(* PLC project Unnamed, Unknown Unnamed 1 *)
(* stored: creationDateTime 2023-03-10T10:37:17, modificationDateTime 2023-03-23T23:20:19 *)

(* SIEMENS AG- Beispielprogramm *)
FUNCTION_BLOCK Bending_Machine_Control
  VAR_INPUT
    IN1 : BOOL;
    IN2 : BOOL;
    IN3 : BOOL;
  END_VAR
  VAR_OUTPUT
    OUT1 : BOOL;
    OUT2 : BOOL;
    OUT3 : BOOL;
  END_VAR
  VAR
    PT5s : TIME;
    PT05s : TIME;
    PT1s : TIME;
    TON0 : TON;
    TON1 : TON;
    TON2 : TON;
    TOF0 : TOF;
    TON3 : TON;
    RS0 : RS;
  END_VAR
  VAR  (* added by the conversion: wires and edge detectors of the diagram *)
    _AND8_OUT : BOOL;
    _AND12_OUT : BOOL;
    _AND18_OUT : BOOL;
    _AND19_OUT : BOOL;
  END_VAR

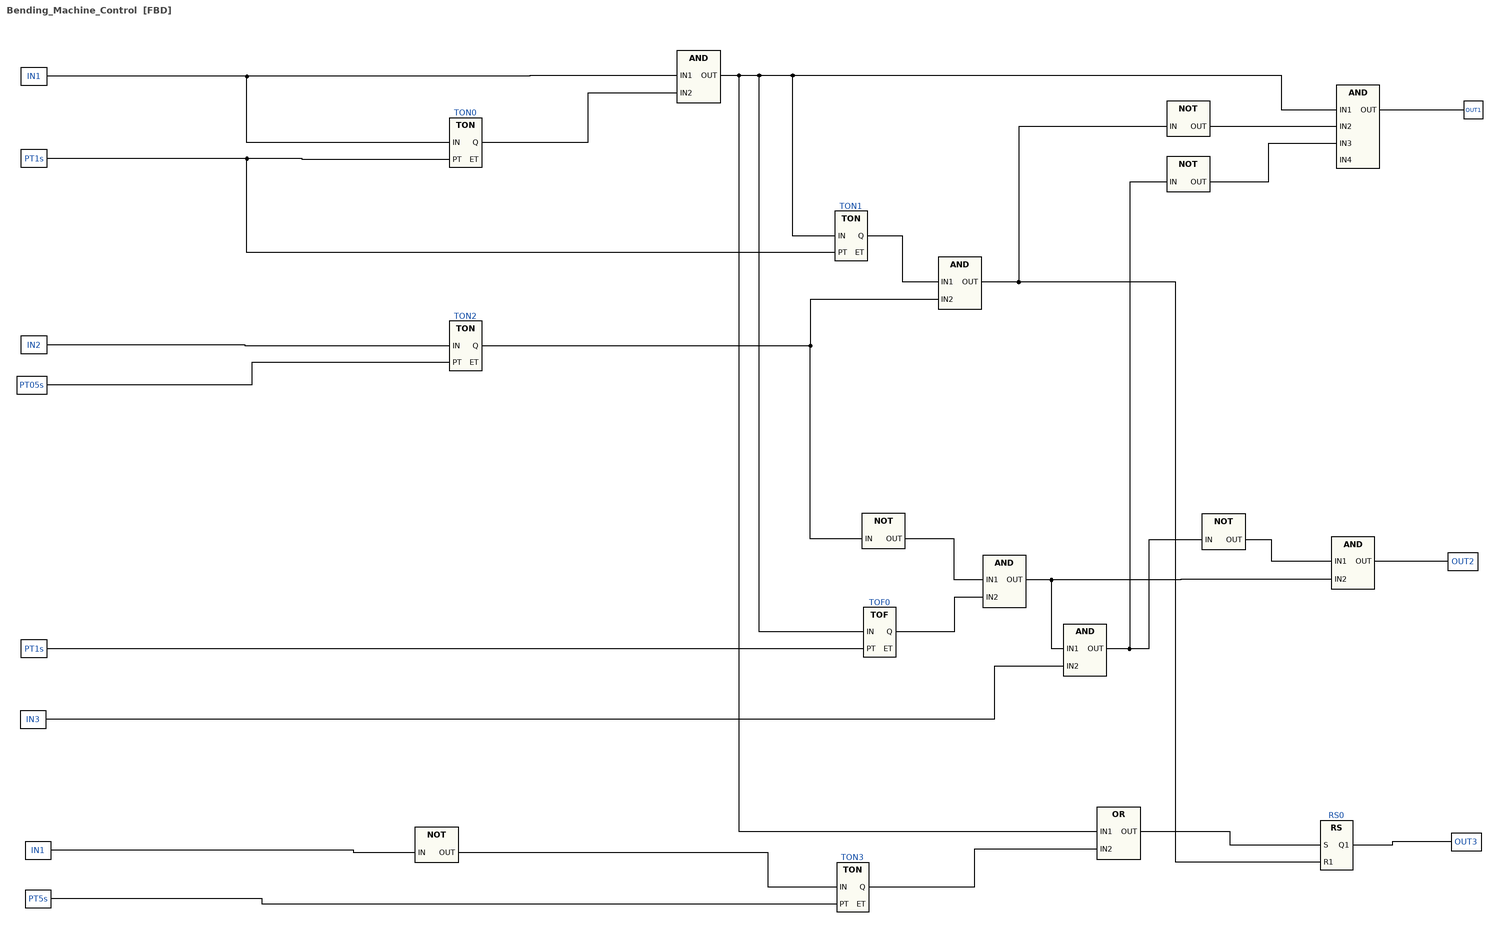
(* FBD diagram, written out as Structured Text *)
TON0(IN := IN1, PT := PT1s);
_AND8_OUT := IN1 AND TON0.Q;
TON1(IN := _AND8_OUT, PT := PT1s);
TON2(IN := IN2, PT := PT05s);
_AND12_OUT := TON1.Q AND TON2.Q;
TOF0(IN := _AND8_OUT, PT := PT1s);
_AND18_OUT := NOT TON2.Q AND TOF0.Q;
_AND19_OUT := _AND18_OUT AND IN3;
OUT1 := AND(IN1 := _AND8_OUT, IN2 := NOT _AND12_OUT, IN3 := NOT _AND19_OUT);
OUT2 := NOT _AND19_OUT AND _AND18_OUT;
TON3(IN := NOT IN1, PT := PT5s);
RS0(S := _AND8_OUT OR TON3.Q, R1 := _AND12_OUT);
OUT3 := RS0.Q1;
END_FUNCTION_BLOCK

CONFIGURATION config
  RESOURCE resource1 ON PLC
  END_RESOURCE
END_CONFIGURATION
